FUNCTION_BLOCK Idle_State  IMPLEMENTS ITF_State
VAR_INPUT
END_VAR
VAR_OUTPUT
END_VAR
VAR
	pPML_Base : POINTER TO PML_StatePattern_Base;
	_stateMachine : IPmlStateMachine;
END_VAR

METHOD Cycle : BOOL
VAR_INPUT
END_VAR
IF _stateMachine.GetCurrentState() = E_PMLState.ePMLState_Starting THEN
	pPML_Base^.SetState(pPML_Base^.starting);
END_IF
END_METHOD

METHOD FB_init : BOOL
VAR_INPUT
	bInitRetains : BOOL; // if TRUE, the retain variables are initialized (warm start / cold start)
	bInCopyCode : BOOL;  // if TRUE, the instance afterwards gets moved into the copy code (online change)
	pPML_Base : POINTER TO PML_StatePattern_Base;
	statemachine : IPmlStateMachine;
END_VAR
_stateMachine := statemachine;
THIS^.pPML_Base := pPML_Base;
END_METHOD

END_FUNCTION_BLOCK

(* stored: Version 1.1.0.1, ProductVersion 3.1.4024.11
   POU Idle_State: Id {7dd3493a-af27-400c-95e9-54528a424b7f}, SpecialFunc None
   Method Cycle: Id {08cf2592-dd1a-4742-9586-4d17f06723f4}
   Method FB_init: Id {02d6e4c9-2d21-4223-b8b8-ec21968f85fd} *)
